(* Logix 5000 project; controller HP_SSC01hv vendor 1 type 14 code 158 rev 32.11; software revision 32.03; part 4 of 15 *)
(* tags used below, declared in another part *)
   A_C1_0422 : ALIAS FOR C1_Warning.22;
   A_C1_0423 : ALIAS FOR C1_Warning.23;
   A_C1_0425 : ALIAS FOR C1_Warning.25;
   A_C1_0426 : ALIAS FOR C1_Warning.26;
   C1_32HourTimers : TIMER[8];
   C1_ActualPositionMOD60 : REAL;
   C1_All_DLY_OK : BOOL;
   C1_Brake_Daily_ok : BOOL;
   C1_BrakeReleaseSelected : BOOL;
   C1_BrakeTestExpireTime : DINT;
   C1_BrakeTestExpireTimeTemp : DINT;
   C1_BrakeTestFailed : BOOL;
   C1_BrakeTestMessageNumber : DINT;
   C1_BrakeTestSelected : BOOL;
   C1_BrakeTestSequence : DINT;
   C1_BrakeTestWarning : BOOL;
   C1_DistanceToEvac : REAL;
   C1_Dump_OK : BOOL;
   C1_DumpValveReleaseSelected : BOOL;
   C1_DumpValveTestExpireTime : DINT;
   C1_DumpValveTestExpireTimeTemp : DINT;
   C1_DumpValveTestSelected : BOOL;
   C1_DumpValveTestSequence : DINT;
   C1_EvacPosition : REAL;
   C1_EvacPositionMOD60 : REAL;
   C1_ExcecutePBHoldTimer : TIMER;
   C1_FaultStandard : DINT;
   C1_GoNearOnPathDelay : TIMER;
   C1_GoToEvacMAM01 : MOTION_INSTRUCTION;
   C1_GoToOnPathMAM01 : MOTION_INSTRUCTION;
   C1_GoToOnPathMAM02 : MOTION_INSTRUCTION;
   C1_Home_OK : BOOL;
   C1_Homed : BOOL;
   C1_HomeExpireTime : DINT;
   C1_HomeExpireTimeTemp : DINT;
   C1_HomeSequence : DINT;
   C1_JogForwardFastSelected : BOOL;
   C1_JogForwardSlowSelected : BOOL;
   C1_JogReverseFastSelected : BOOL;
   C1_JogReverseSlowSelected : BOOL;
   C1_LubricationMessageNumber : DINT;
   C1_LubricationOnTimer : TIMER;
   C1_LubricationOverrideSelected : BOOL;
   C1_MAFR : MOTION_INSTRUCTION;
   C1_MAG : MOTION_INSTRUCTION;
   C1_MAJDeceleration : REAL;
   C1_MAS : MOTION_INSTRUCTION;
   C1_MASR : MOTION_INSTRUCTION;
   C1_Oiler : ALIAS FOR C1_RIO_AENT:O.Data[2].1;
   C1_OIT_BrakeRelease : BOOL;
   C1_OIT_BrakeReleaseDisplay : BOOL;
   C1_OIT_BrakeTest : BOOL;
   C1_OIT_BrakeTestDisplay : BOOL;
   C1_OIT_Command : DINT;
   C1_OIT_Current : DINT;
   C1_OIT_DumpValveRelease : BOOL;
   C1_OIT_DumpValveReleaseDisplay : BOOL;
   C1_OIT_DumpValveTest : BOOL;
   C1_OIT_DumpValveTestDisplay : BOOL;
   C1_OIT_FaultsExist : BOOL;
   C1_OIT_HomeCountDown : DINT;
   C1_OIT_JogForwardFast : BOOL;
   C1_OIT_JogForwardFastDisplay : BOOL;
   C1_OIT_JogForwardSlow : BOOL;
   C1_OIT_JogForwardSlowDisplay : BOOL;
   C1_OIT_JogReverseFast : BOOL;
   C1_OIT_JogReverseFastDisplay : BOOL;
   C1_OIT_JogReverseSlow : BOOL;
   C1_OIT_JogReverseSlowDisplay : BOOL;
   C1_OIT_JogStopDisplay : BOOL;
   C1_OIT_LubricationOverride : BOOL;
   C1_OIT_LubricationOverrideDisplay : BOOL;
   C1_OIT_PathError : DINT;
   C1_OIT_PathIndicatorHigh : DINT;
   C1_OIT_PathIndicatorLow : DINT;
   C1_OIT_WarningsExist : BOOL;
   C1_OneTryToFixErrorONS : BOOL;
   C1_ONS : DINT;
   C1_RemoteBrakeAndHomeSequence : DINT;
   C1_RemoteBrakeAndHomeSequenceAlarms : DINT;
   C1_RemoteBrakeAndHomeSequenceAlarmTimer : TIMER[32];
   C1_RemoteBrakeAndHomeSequenceONS : BOOL;
   C1_RemoteBrakeTestCMD : BOOL;
   C1_RemoteDumpTestCMD : BOOL;
   C1_RemoteHomeCMD : BOOL;
   C1_RemoteScreenMessageNumber : DINT;
   C1_RemoteSequenceDelay : TIMER[8];
   C1_RevolutionCounter : COUNTER;
   C1_ServoActionStatusOnDelay : TIMER;
   C1_TargetPositionError : REAL;
   C1_TargetPositionErrorTest : REAL;
   C1_Warning : DINT;
   MasterClockCopyMAS_Stop1 : MOTION_INSTRUCTION;
   MasterClockCopyMAS_Stop2 : MOTION_INSTRUCTION;
   MasterClockLocal : AXIS_VIRTUAL;
   none : BOOL;
   RCS_CMD_Auto_TON : TIMER;
   RCS_MasterClockLocalTagetDegrees : REAL;
   S_C1_FaultReset : BOOL;
   S_C1_FaultSafety : DINT;
   S_C1_ModeLocal : BOOL;
   S_C1_ModeRemote : BOOL;
   S_C1_MSTOP_InputOK : BOOL;
   S_C1_NearOnPath : BOOL;
   S_C1_NearOnPathHi : DINT;
   S_C1_NearOnPathLow : DINT;
   S_C1_OffPath : BOOL;
   S_C1_OnPath : BOOL;
   S_C1_PathError : DINT;
   S_RCS_MotionCMD_BrakeTest : BOOL;
   S_RCS_MotionCMD_Evac : BOOL;
   S_RCS_MotionCMD_GoNearOnPath : BOOL;
(* Carousel1, continued *)

ROUTINE C145_Lubrication   (* ladder *)
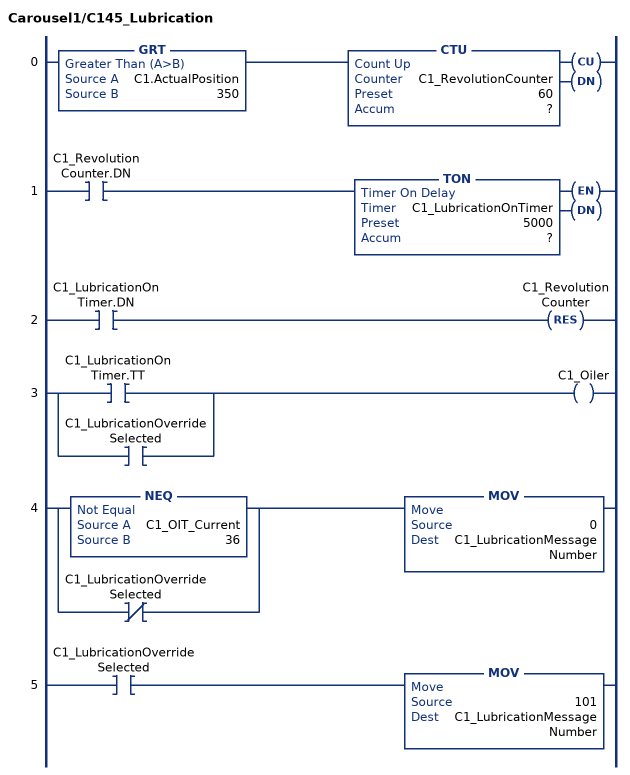
   0: GRT(C1.ActualPosition,350)CTU(C1_RevolutionCounter,?,?);
   1: XIC(C1_RevolutionCounter.DN)TON(C1_LubricationOnTimer,?,?);
   2: XIC(C1_LubricationOnTimer.DN)RES(C1_RevolutionCounter);
   3: [XIC(C1_LubricationOnTimer.TT) ,XIC(C1_LubricationOverrideSelected) ]OTE(C1_Oiler);
   4: [NEQ(C1_OIT_Current,36) ,XIO(C1_LubricationOverrideSelected) ]MOV(0,C1_LubricationMessageNumber);
   5: XIC(C1_LubricationOverrideSelected)MOV(101,C1_LubricationMessageNumber);
END_ROUTINE

ROUTINE C150_OIT   (* ladder *)
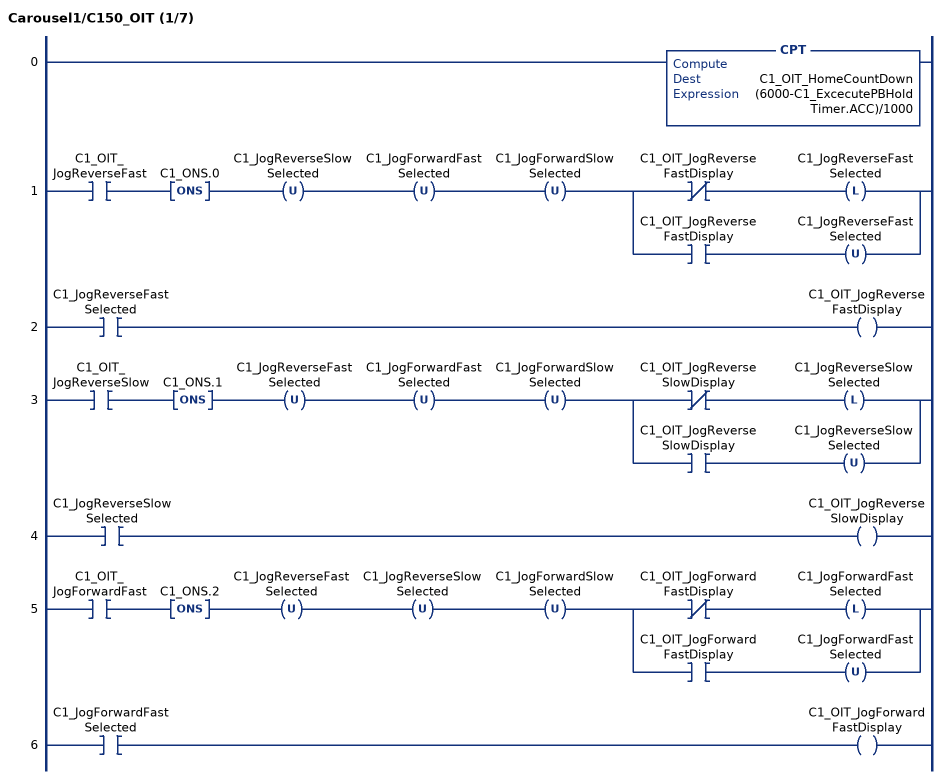
   0: CPT(C1_OIT_HomeCountDown,(6000-C1_ExcecutePBHoldTimer.ACC)/1000);
   1: XIC(C1_OIT_JogReverseFast)ONS(C1_ONS.0)OTU(C1_JogReverseSlowSelected)OTU(C1_JogForwardFastSelected)OTU(C1_JogForwardSlowSelected)[XIO(C1_OIT_JogReverseFastDisplay) OTL(C1_JogReverseFastSelected) ,XIC(C1_OIT_JogReverseFastDisplay) OTU(C1_JogReverseFastSelected) ];
   2: XIC(C1_JogReverseFastSelected)OTE(C1_OIT_JogReverseFastDisplay);
   3: XIC(C1_OIT_JogReverseSlow)ONS(C1_ONS.1)OTU(C1_JogReverseFastSelected)OTU(C1_JogForwardFastSelected)OTU(C1_JogForwardSlowSelected)[XIO(C1_OIT_JogReverseSlowDisplay) OTL(C1_JogReverseSlowSelected) ,XIC(C1_OIT_JogReverseSlowDisplay) OTU(C1_JogReverseSlowSelected) ];
   4: XIC(C1_JogReverseSlowSelected)OTE(C1_OIT_JogReverseSlowDisplay);
   5: XIC(C1_OIT_JogForwardFast)ONS(C1_ONS.2)OTU(C1_JogReverseFastSelected)OTU(C1_JogReverseSlowSelected)OTU(C1_JogForwardSlowSelected)[XIO(C1_OIT_JogForwardFastDisplay) OTL(C1_JogForwardFastSelected) ,XIC(C1_OIT_JogForwardFastDisplay) OTU(C1_JogForwardFastSelected) ];
   6: XIC(C1_JogForwardFastSelected)OTE(C1_OIT_JogForwardFastDisplay);
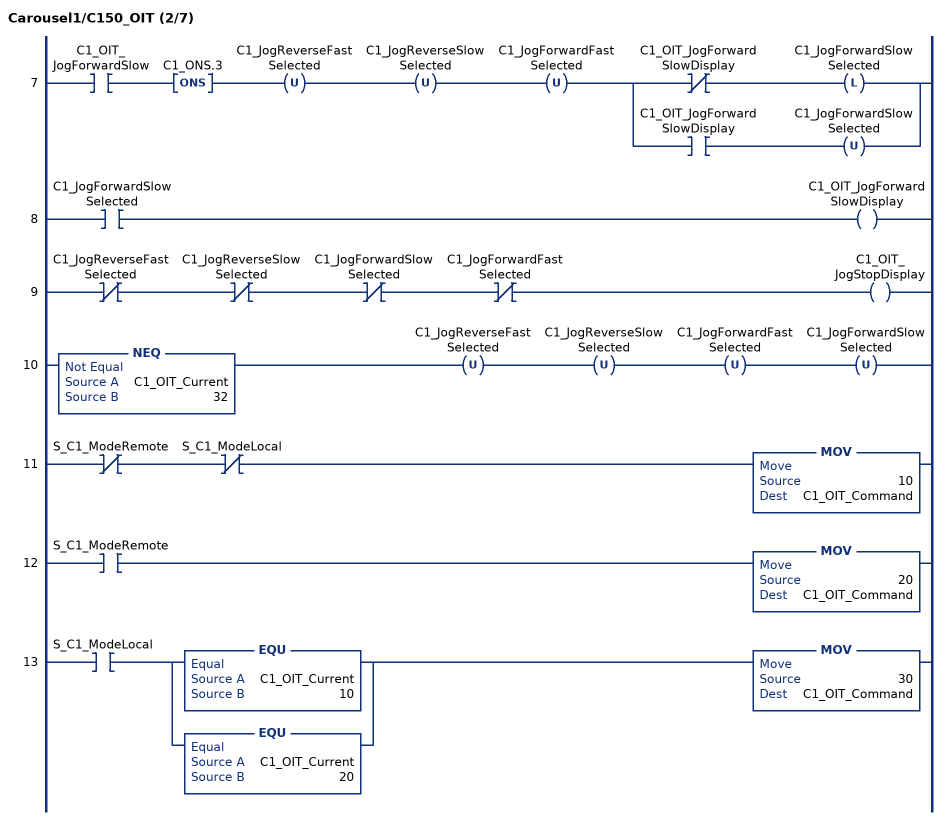
   7: XIC(C1_OIT_JogForwardSlow)ONS(C1_ONS.3)OTU(C1_JogReverseFastSelected)OTU(C1_JogReverseSlowSelected)OTU(C1_JogForwardFastSelected)[XIO(C1_OIT_JogForwardSlowDisplay) OTL(C1_JogForwardSlowSelected) ,XIC(C1_OIT_JogForwardSlowDisplay) OTU(C1_JogForwardSlowSelected) ];
   8: XIC(C1_JogForwardSlowSelected)OTE(C1_OIT_JogForwardSlowDisplay);
   9: XIO(C1_JogReverseFastSelected)XIO(C1_JogReverseSlowSelected)XIO(C1_JogForwardSlowSelected)XIO(C1_JogForwardFastSelected)OTE(C1_OIT_JogStopDisplay);
   10: NEQ(C1_OIT_Current,32)OTU(C1_JogReverseFastSelected)OTU(C1_JogReverseSlowSelected)OTU(C1_JogForwardFastSelected)OTU(C1_JogForwardSlowSelected);
   11: XIO(S_C1_ModeRemote)XIO(S_C1_ModeLocal)MOV(10,C1_OIT_Command);
   12: XIC(S_C1_ModeRemote)MOV(20,C1_OIT_Command);
   13: XIC(S_C1_ModeLocal)[EQU(C1_OIT_Current,10) ,EQU(C1_OIT_Current,20) ]MOV(30,C1_OIT_Command);
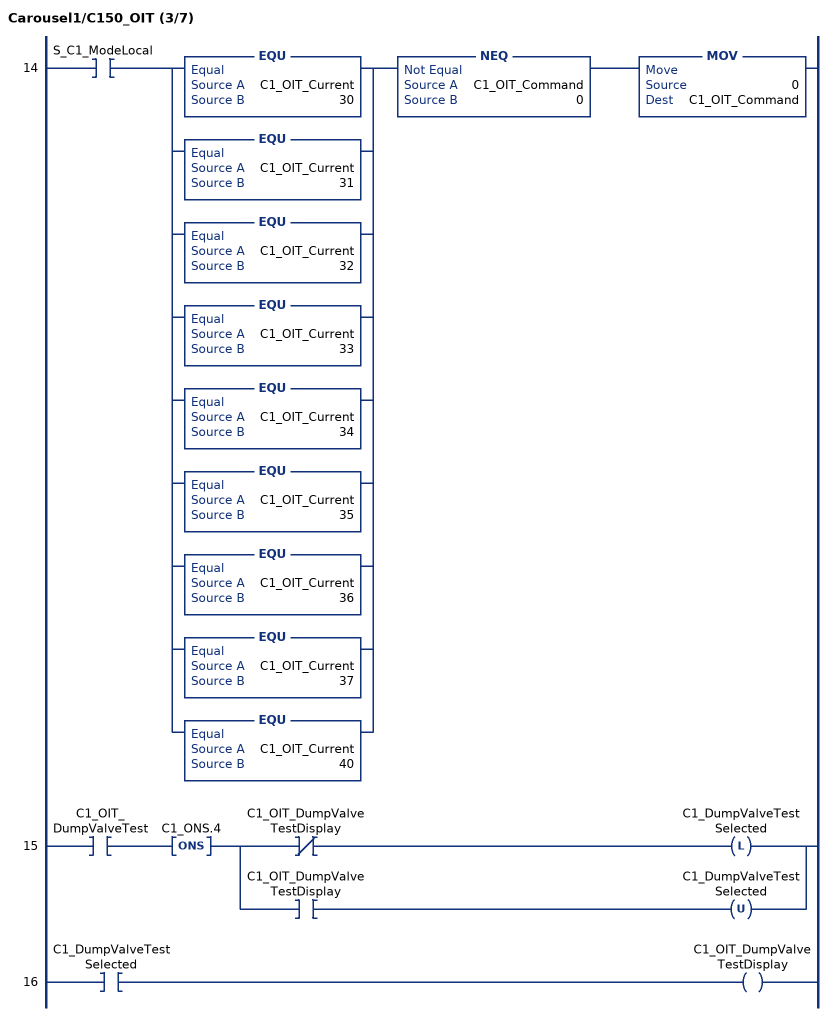
   14: XIC(S_C1_ModeLocal)[EQU(C1_OIT_Current,30) ,EQU(C1_OIT_Current,31) ,EQU(C1_OIT_Current,32) ,EQU(C1_OIT_Current,33) ,EQU(C1_OIT_Current,34) ,EQU(C1_OIT_Current,35) ,EQU(C1_OIT_Current,36) ,EQU(C1_OIT_Current,37) ,EQU(C1_OIT_Current,40) ]NEQ(C1_OIT_Command,0)MOV(0,C1_OIT_Command);
   15: XIC(C1_OIT_DumpValveTest)ONS(C1_ONS.4)[XIO(C1_OIT_DumpValveTestDisplay) OTL(C1_DumpValveTestSelected) ,XIC(C1_OIT_DumpValveTestDisplay) OTU(C1_DumpValveTestSelected) ];
   16: XIC(C1_DumpValveTestSelected)OTE(C1_OIT_DumpValveTestDisplay);
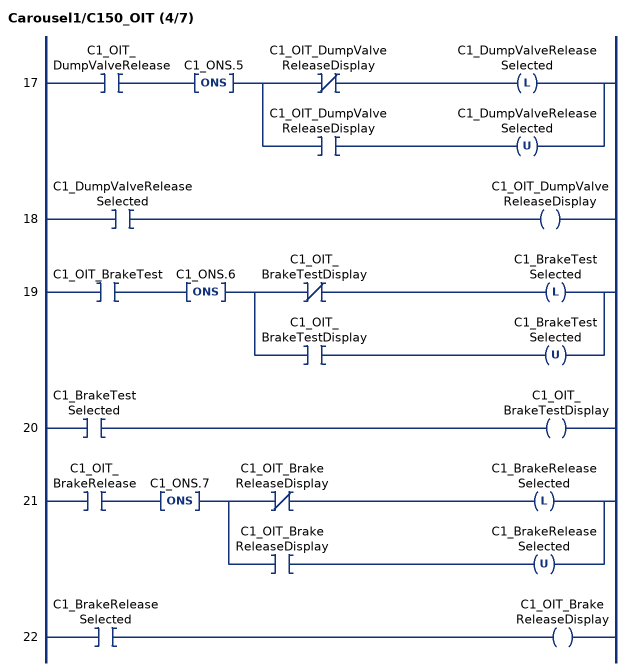
   17: XIC(C1_OIT_DumpValveRelease)ONS(C1_ONS.5)[XIO(C1_OIT_DumpValveReleaseDisplay) OTL(C1_DumpValveReleaseSelected) ,XIC(C1_OIT_DumpValveReleaseDisplay) OTU(C1_DumpValveReleaseSelected) ];
   18: XIC(C1_DumpValveReleaseSelected)OTE(C1_OIT_DumpValveReleaseDisplay);
   19: XIC(C1_OIT_BrakeTest)ONS(C1_ONS.6)[XIO(C1_OIT_BrakeTestDisplay) OTL(C1_BrakeTestSelected) ,XIC(C1_OIT_BrakeTestDisplay) OTU(C1_BrakeTestSelected) ];
   20: XIC(C1_BrakeTestSelected)OTE(C1_OIT_BrakeTestDisplay);
   21: XIC(C1_OIT_BrakeRelease)ONS(C1_ONS.7)[XIO(C1_OIT_BrakeReleaseDisplay) OTL(C1_BrakeReleaseSelected) ,XIC(C1_OIT_BrakeReleaseDisplay) OTU(C1_BrakeReleaseSelected) ];
   22: XIC(C1_BrakeReleaseSelected)OTE(C1_OIT_BrakeReleaseDisplay);
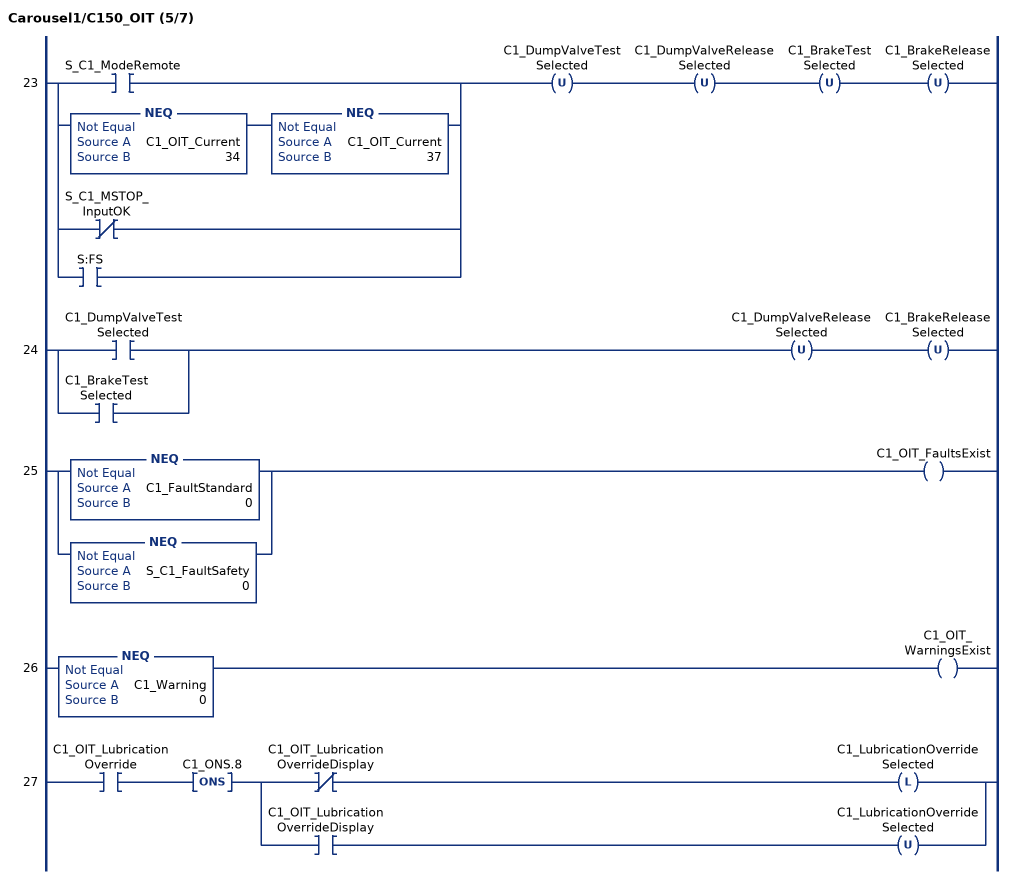
   23: [XIC(S_C1_ModeRemote) ,NEQ(C1_OIT_Current,34) NEQ(C1_OIT_Current,37) ,XIO(S_C1_MSTOP_InputOK) ,XIC(S:FS) ]OTU(C1_DumpValveTestSelected)OTU(C1_DumpValveReleaseSelected)OTU(C1_BrakeTestSelected)OTU(C1_BrakeReleaseSelected);
   24: [XIC(C1_DumpValveTestSelected) ,XIC(C1_BrakeTestSelected) ]OTU(C1_DumpValveReleaseSelected)OTU(C1_BrakeReleaseSelected);
   25: [NEQ(C1_FaultStandard,0) ,NEQ(S_C1_FaultSafety,0) ]OTE(C1_OIT_FaultsExist);
   26: NEQ(C1_Warning,0)OTE(C1_OIT_WarningsExist);
   27: XIC(C1_OIT_LubricationOverride)ONS(C1_ONS.8)[XIO(C1_OIT_LubricationOverrideDisplay) OTL(C1_LubricationOverrideSelected) ,XIC(C1_OIT_LubricationOverrideDisplay) OTU(C1_LubricationOverrideSelected) ];
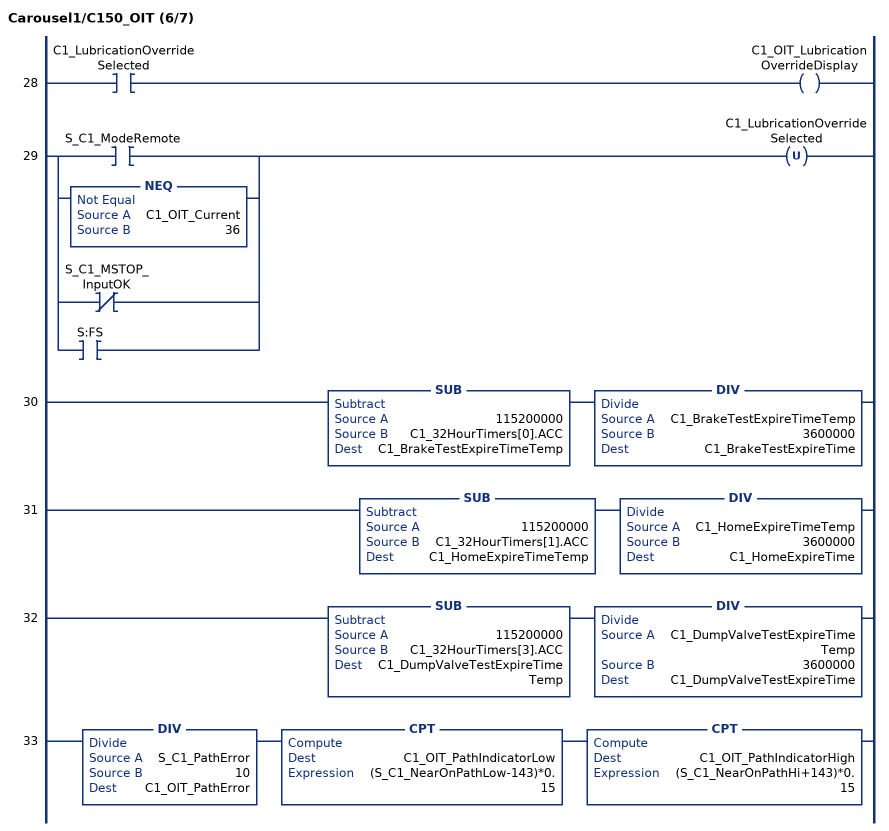
   28: XIC(C1_LubricationOverrideSelected)OTE(C1_OIT_LubricationOverrideDisplay);
   29: [XIC(S_C1_ModeRemote) ,NEQ(C1_OIT_Current,36) ,XIO(S_C1_MSTOP_InputOK) ,XIC(S:FS) ]OTU(C1_LubricationOverrideSelected);
   30: SUB(115200000,C1_32HourTimers[0].ACC,C1_BrakeTestExpireTimeTemp)DIV(C1_BrakeTestExpireTimeTemp,3600000,C1_BrakeTestExpireTime);
   31: SUB(115200000,C1_32HourTimers[1].ACC,C1_HomeExpireTimeTemp)DIV(C1_HomeExpireTimeTemp,3600000,C1_HomeExpireTime);
   32: SUB(115200000,C1_32HourTimers[3].ACC,C1_DumpValveTestExpireTimeTemp)DIV(C1_DumpValveTestExpireTimeTemp,3600000,C1_DumpValveTestExpireTime);
   33: DIV(S_C1_PathError,10,C1_OIT_PathError)CPT(C1_OIT_PathIndicatorLow,(S_C1_NearOnPathLow-143)*0.15)CPT(C1_OIT_PathIndicatorHigh,(S_C1_NearOnPathHi+143)*0.15);
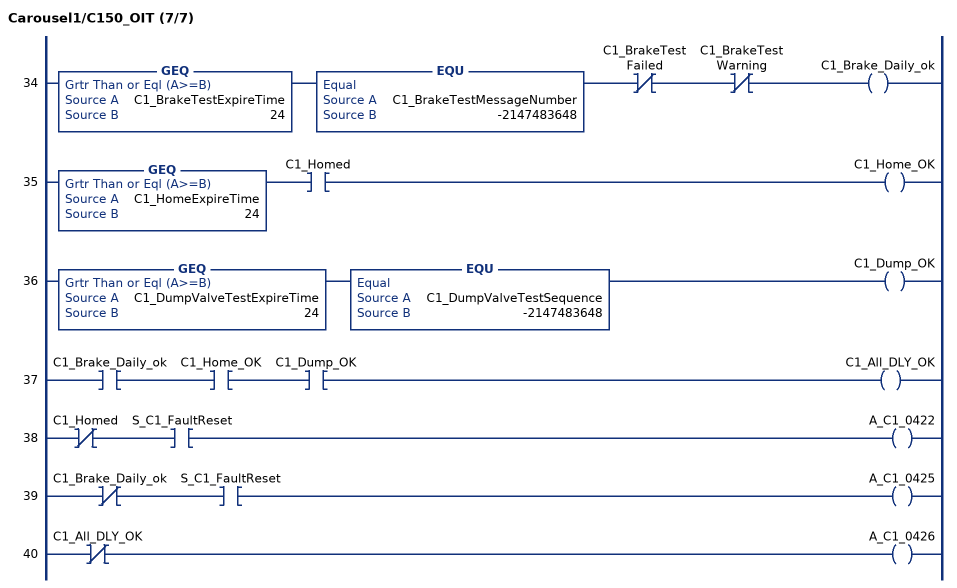
   34: GEQ(C1_BrakeTestExpireTime,24)EQU(C1_BrakeTestMessageNumber,-2147483648)XIO(C1_BrakeTestFailed)XIO(C1_BrakeTestWarning)OTE(C1_Brake_Daily_ok);
   35: GEQ(C1_HomeExpireTime,24)XIC(C1_Homed)OTE(C1_Home_OK);
   36: GEQ(C1_DumpValveTestExpireTime,24)EQU(C1_DumpValveTestSequence,-2147483648)OTE(C1_Dump_OK);
   37: XIC(C1_Brake_Daily_ok)XIC(C1_Home_OK)XIC(C1_Dump_OK)OTE(C1_All_DLY_OK);
   38: XIO(C1_Homed)XIC(S_C1_FaultReset)OTE(A_C1_0422);
   39: XIO(C1_Brake_Daily_ok)XIC(S_C1_FaultReset)OTE(A_C1_0425);
   40: XIO(C1_All_DLY_OK)OTE(A_C1_0426);
END_ROUTINE

ROUTINE C155_Remote   (* ladder *)
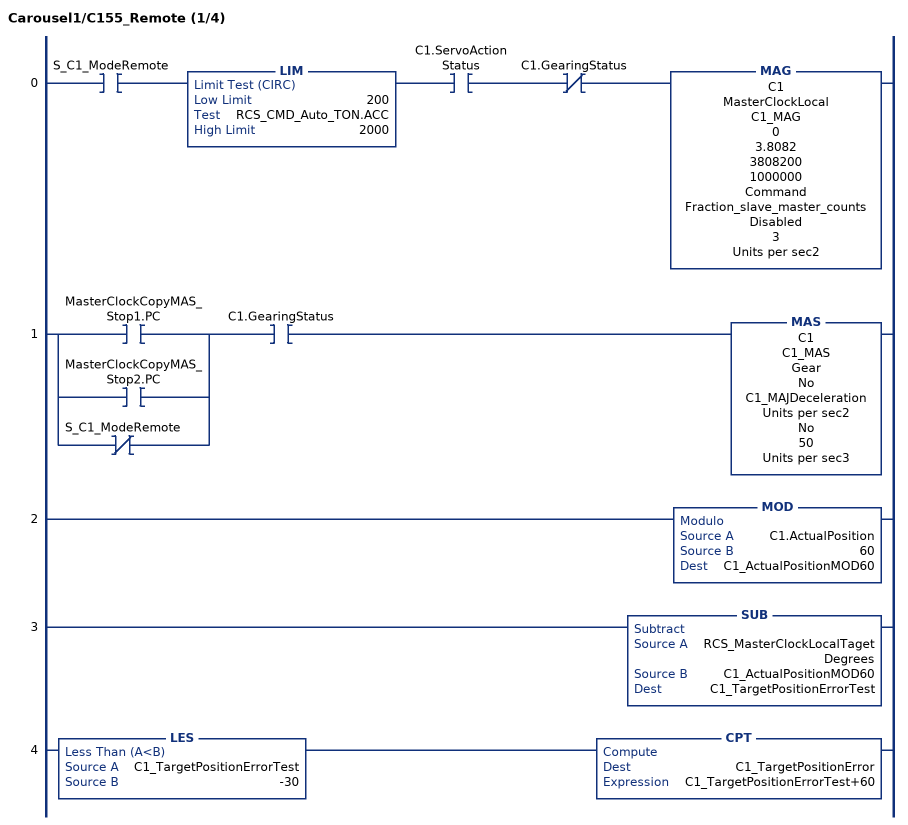
   0: XIC(S_C1_ModeRemote)LIM(200,RCS_CMD_Auto_TON.ACC,2000)XIC(C1.ServoActionStatus)XIO(C1.GearingStatus)MAG(C1,MasterClockLocal,C1_MAG,0,3.8082,3808200,1000000,Command,Fraction_slave_master_counts,Disabled,3,Units per sec2);
   1: [XIC(MasterClockCopyMAS_Stop1.PC) ,XIC(MasterClockCopyMAS_Stop2.PC) ,XIO(S_C1_ModeRemote) ]XIC(C1.GearingStatus)MAS(C1,C1_MAS,Gear,No,C1_MAJDeceleration,Units per sec2,No,50,Units per sec3);
   2: MOD(C1.ActualPosition,60,C1_ActualPositionMOD60);
   3: SUB(RCS_MasterClockLocalTagetDegrees,C1_ActualPositionMOD60,C1_TargetPositionErrorTest);
   4: LES(C1_TargetPositionErrorTest,-30)CPT(C1_TargetPositionError,C1_TargetPositionErrorTest+60);
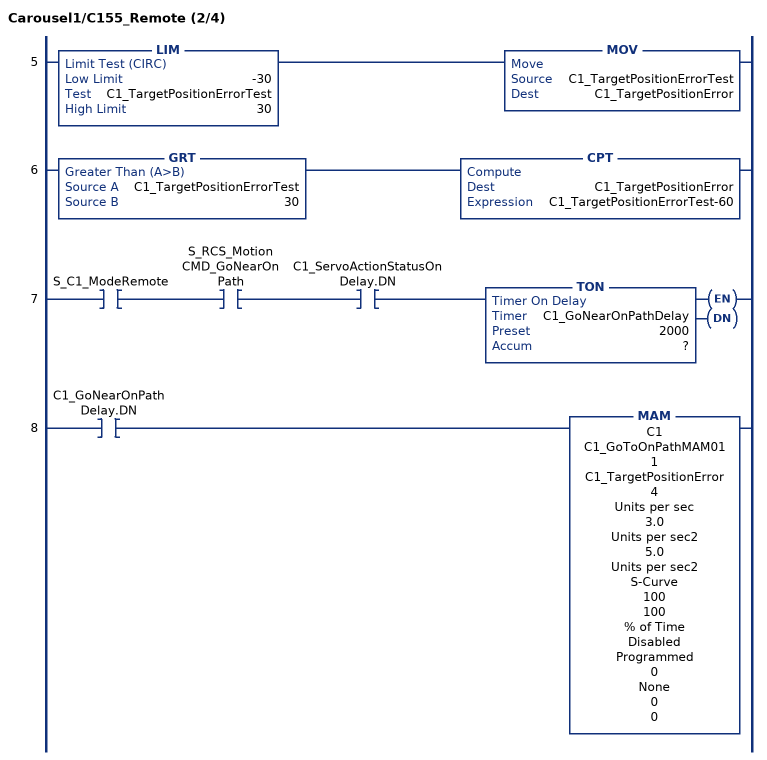
   5: LIM(-30,C1_TargetPositionErrorTest,30)MOV(C1_TargetPositionErrorTest,C1_TargetPositionError);
   6: GRT(C1_TargetPositionErrorTest,30)CPT(C1_TargetPositionError,C1_TargetPositionErrorTest-60);
   7: XIC(S_C1_ModeRemote)XIC(S_RCS_MotionCMD_GoNearOnPath)XIC(C1_ServoActionStatusOnDelay.DN)TON(C1_GoNearOnPathDelay,?,?);
   8: XIC(C1_GoNearOnPathDelay.DN)MAM(C1,C1_GoToOnPathMAM01,1,C1_TargetPositionError,4,Units per sec,3.0,Units per sec2,5.0,Units per sec2,S-Curve,100,100,% of Time,Disabled,Programmed,0,None,0,0);
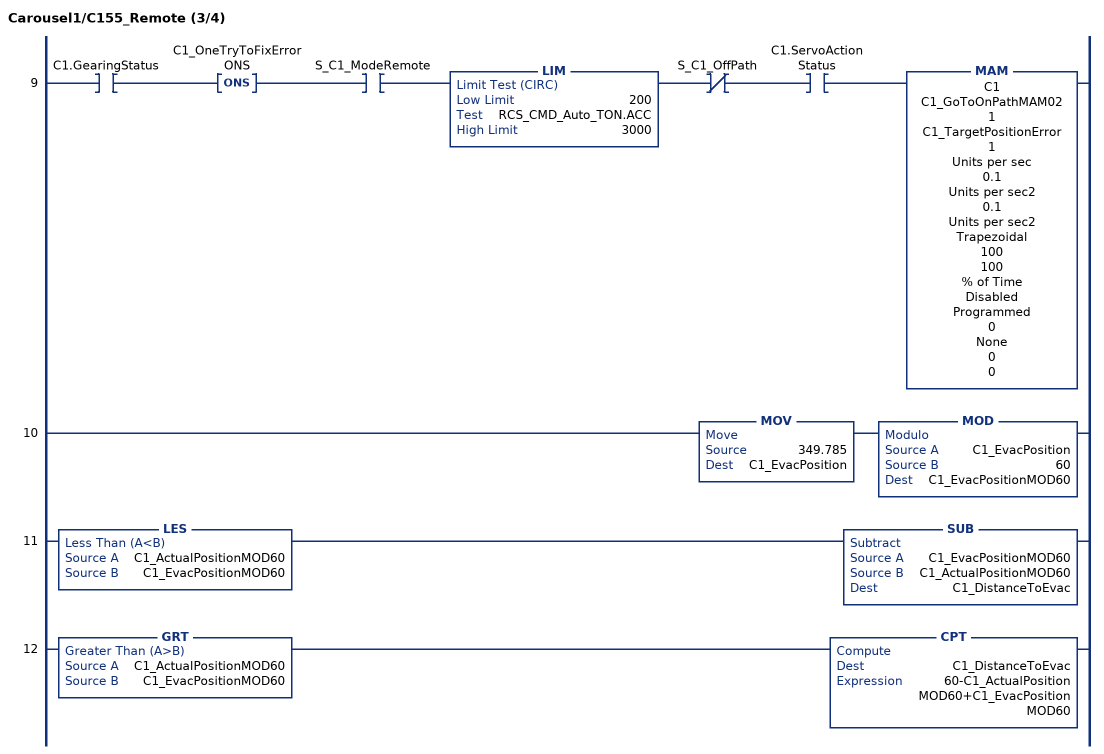
   9: XIC(C1.GearingStatus)ONS(C1_OneTryToFixErrorONS)XIC(S_C1_ModeRemote)LIM(200,RCS_CMD_Auto_TON.ACC,3000)XIO(S_C1_OffPath)XIC(C1.ServoActionStatus)MAM(C1,C1_GoToOnPathMAM02,1,C1_TargetPositionError,1,Units per sec,0.1,Units per sec2,0.1,Units per sec2,Trapezoidal,100,100,% of Time,Disabled,Programmed,0,None,0,0);
   10: MOV(349.785,C1_EvacPosition)MOD(C1_EvacPosition,60,C1_EvacPositionMOD60);
   11: LES(C1_ActualPositionMOD60,C1_EvacPositionMOD60)SUB(C1_EvacPositionMOD60,C1_ActualPositionMOD60,C1_DistanceToEvac);
   12: GRT(C1_ActualPositionMOD60,C1_EvacPositionMOD60)CPT(C1_DistanceToEvac,60-C1_ActualPositionMOD60+C1_EvacPositionMOD60);
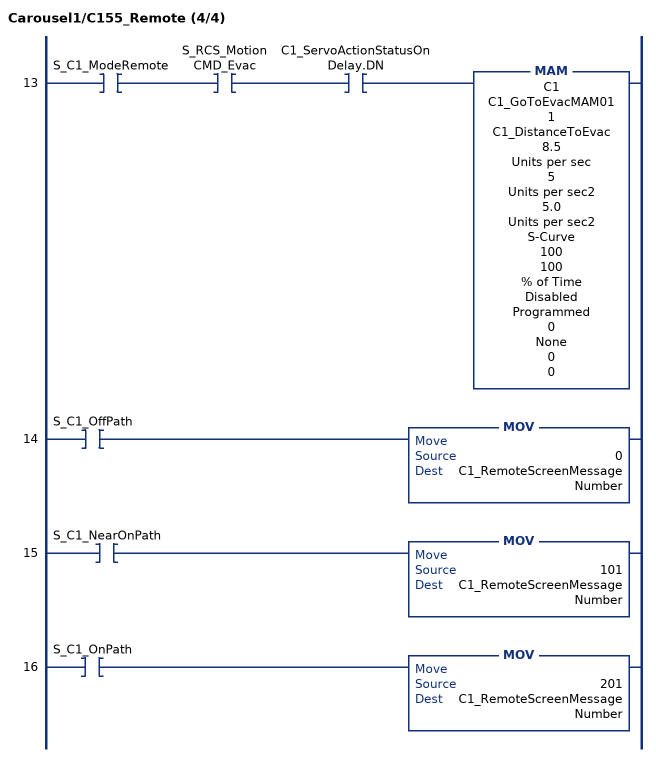
   13: XIC(S_C1_ModeRemote)XIC(S_RCS_MotionCMD_Evac)XIC(C1_ServoActionStatusOnDelay.DN)MAM(C1,C1_GoToEvacMAM01,1,C1_DistanceToEvac,8.5,Units per sec,5,Units per sec2,5.0,Units per sec2,S-Curve,100,100,% of Time,Disabled,Programmed,0,None,0,0);
   14: XIC(S_C1_OffPath)MOV(0,C1_RemoteScreenMessageNumber);
   15: XIC(S_C1_NearOnPath)MOV(101,C1_RemoteScreenMessageNumber);
   16: XIC(S_C1_OnPath)MOV(201,C1_RemoteScreenMessageNumber);
END_ROUTINE

ROUTINE C160_RemoteBrakeAndHome   (* ladder *)
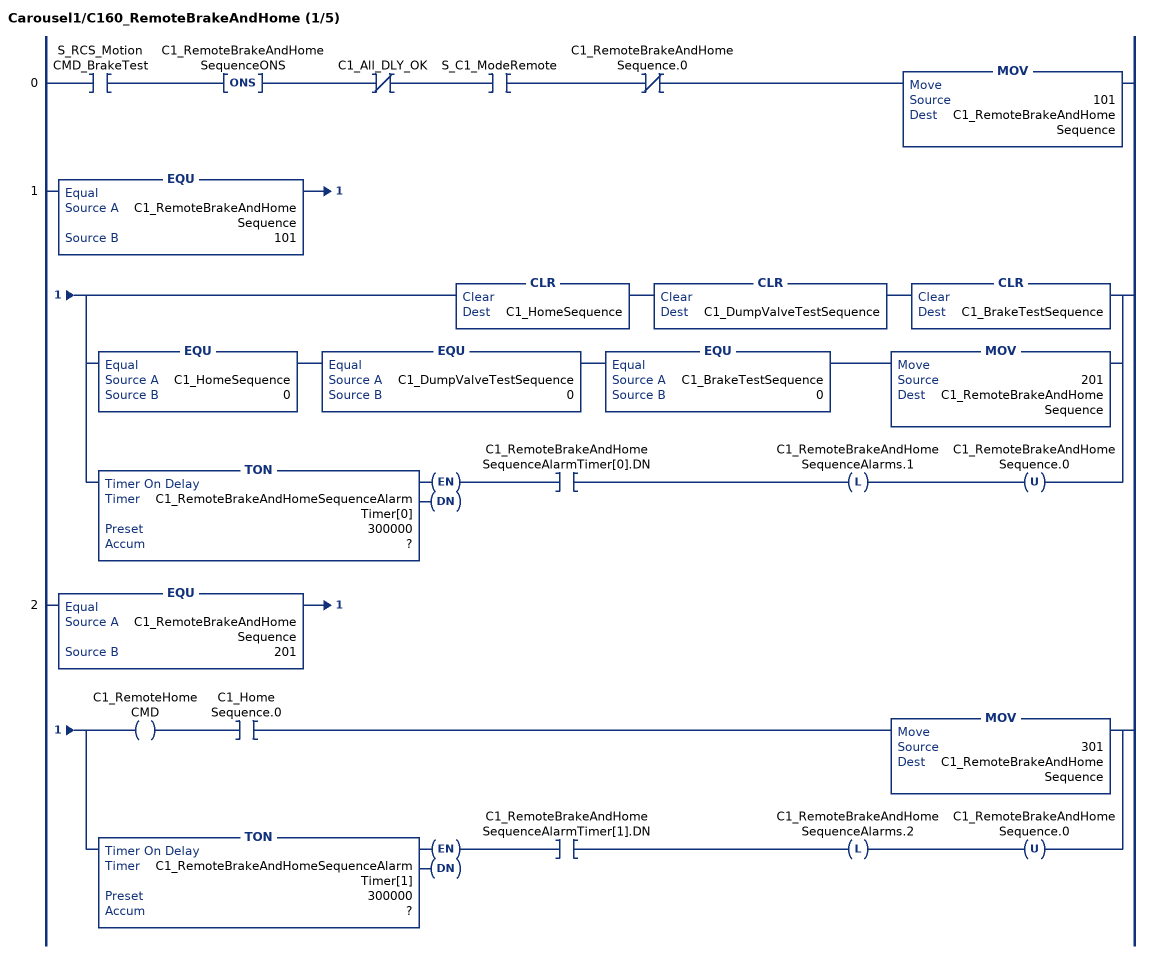
   0: XIC(S_RCS_MotionCMD_BrakeTest)ONS(C1_RemoteBrakeAndHomeSequenceONS)XIO(C1_All_DLY_OK)XIC(S_C1_ModeRemote)XIO(C1_RemoteBrakeAndHomeSequence.0)MOV(101,C1_RemoteBrakeAndHomeSequence);
   1: EQU(C1_RemoteBrakeAndHomeSequence,101)[CLR(C1_HomeSequence) CLR(C1_DumpValveTestSequence) CLR(C1_BrakeTestSequence) ,EQU(C1_HomeSequence,0) EQU(C1_DumpValveTestSequence,0) EQU(C1_BrakeTestSequence,0) MOV(201,C1_RemoteBrakeAndHomeSequence) ,TON(C1_RemoteBrakeAndHomeSequenceAlarmTimer[0],?,?) XIC(C1_RemoteBrakeAndHomeSequenceAlarmTimer[0].DN) OTL(C1_RemoteBrakeAndHomeSequenceAlarms.1) OTU(C1_RemoteBrakeAndHomeSequence.0) ];
   2: EQU(C1_RemoteBrakeAndHomeSequence,201)[OTE(C1_RemoteHomeCMD) XIC(C1_HomeSequence.0) MOV(301,C1_RemoteBrakeAndHomeSequence) ,TON(C1_RemoteBrakeAndHomeSequenceAlarmTimer[1],?,?) XIC(C1_RemoteBrakeAndHomeSequenceAlarmTimer[1].DN) OTL(C1_RemoteBrakeAndHomeSequenceAlarms.2) OTU(C1_RemoteBrakeAndHomeSequence.0) ];
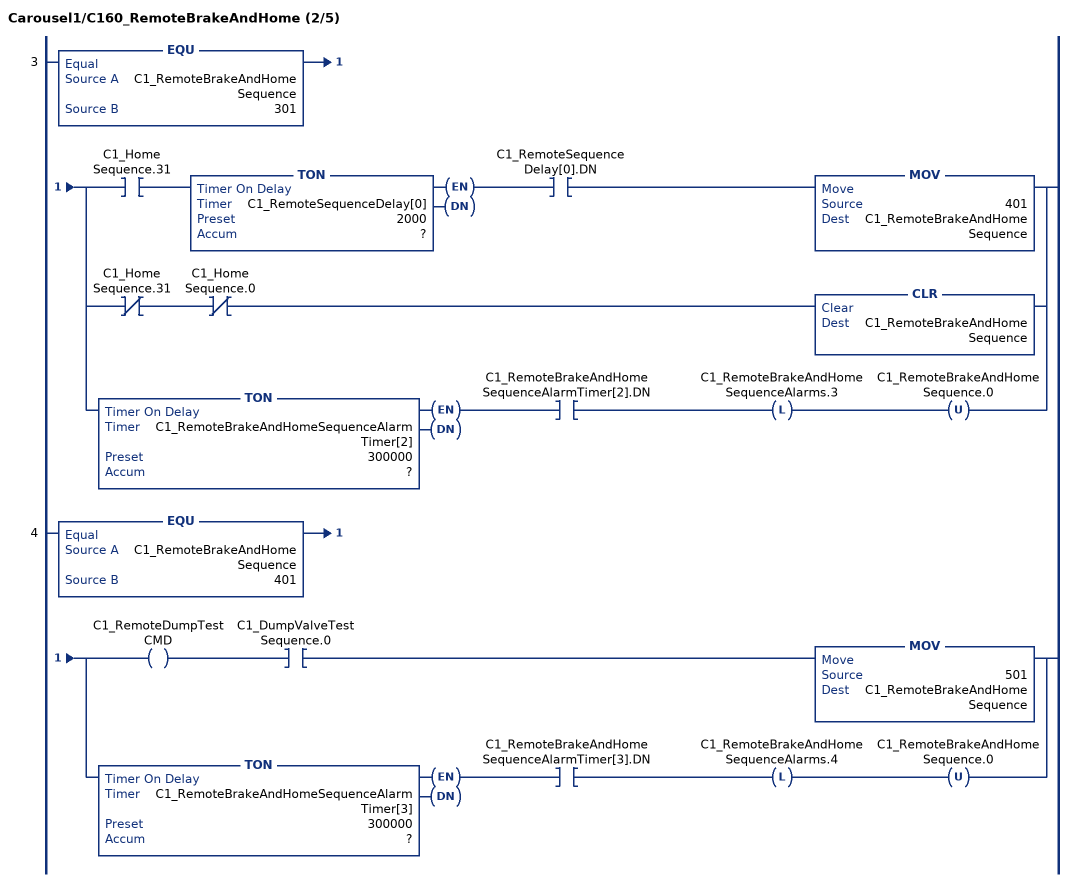
   3: EQU(C1_RemoteBrakeAndHomeSequence,301)[XIC(C1_HomeSequence.31) TON(C1_RemoteSequenceDelay[0],?,?) XIC(C1_RemoteSequenceDelay[0].DN) MOV(401,C1_RemoteBrakeAndHomeSequence) ,XIO(C1_HomeSequence.31) XIO(C1_HomeSequence.0) CLR(C1_RemoteBrakeAndHomeSequence) ,TON(C1_RemoteBrakeAndHomeSequenceAlarmTimer[2],?,?) XIC(C1_RemoteBrakeAndHomeSequenceAlarmTimer[2].DN) OTL(C1_RemoteBrakeAndHomeSequenceAlarms.3) OTU(C1_RemoteBrakeAndHomeSequence.0) ];
   4: EQU(C1_RemoteBrakeAndHomeSequence,401)[OTE(C1_RemoteDumpTestCMD) XIC(C1_DumpValveTestSequence.0) MOV(501,C1_RemoteBrakeAndHomeSequence) ,TON(C1_RemoteBrakeAndHomeSequenceAlarmTimer[3],?,?) XIC(C1_RemoteBrakeAndHomeSequenceAlarmTimer[3].DN) OTL(C1_RemoteBrakeAndHomeSequenceAlarms.4) OTU(C1_RemoteBrakeAndHomeSequence.0) ];
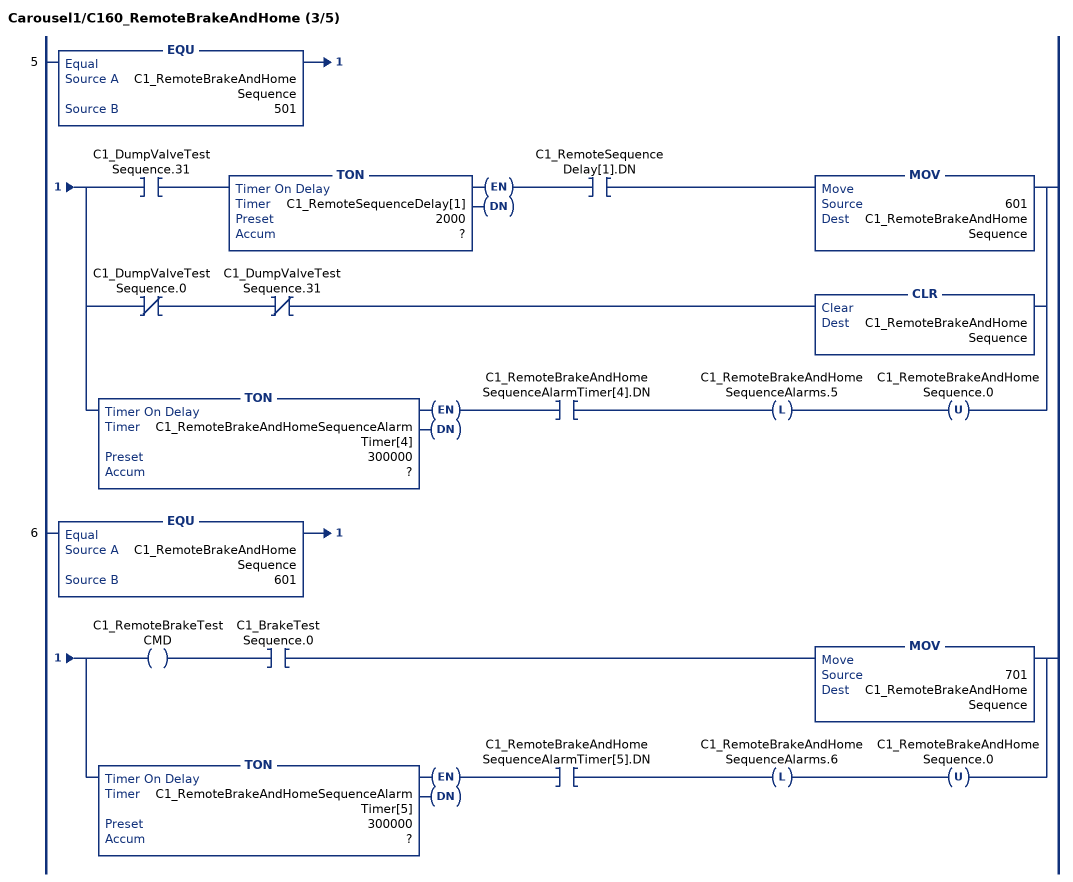
   5: EQU(C1_RemoteBrakeAndHomeSequence,501)[XIC(C1_DumpValveTestSequence.31) TON(C1_RemoteSequenceDelay[1],?,?) XIC(C1_RemoteSequenceDelay[1].DN) MOV(601,C1_RemoteBrakeAndHomeSequence) ,XIO(C1_DumpValveTestSequence.0) XIO(C1_DumpValveTestSequence.31) CLR(C1_RemoteBrakeAndHomeSequence) ,TON(C1_RemoteBrakeAndHomeSequenceAlarmTimer[4],?,?) XIC(C1_RemoteBrakeAndHomeSequenceAlarmTimer[4].DN) OTL(C1_RemoteBrakeAndHomeSequenceAlarms.5) OTU(C1_RemoteBrakeAndHomeSequence.0) ];
   6: EQU(C1_RemoteBrakeAndHomeSequence,601)[OTE(C1_RemoteBrakeTestCMD) XIC(C1_BrakeTestSequence.0) MOV(701,C1_RemoteBrakeAndHomeSequence) ,TON(C1_RemoteBrakeAndHomeSequenceAlarmTimer[5],?,?) XIC(C1_RemoteBrakeAndHomeSequenceAlarmTimer[5].DN) OTL(C1_RemoteBrakeAndHomeSequenceAlarms.6) OTU(C1_RemoteBrakeAndHomeSequence.0) ];
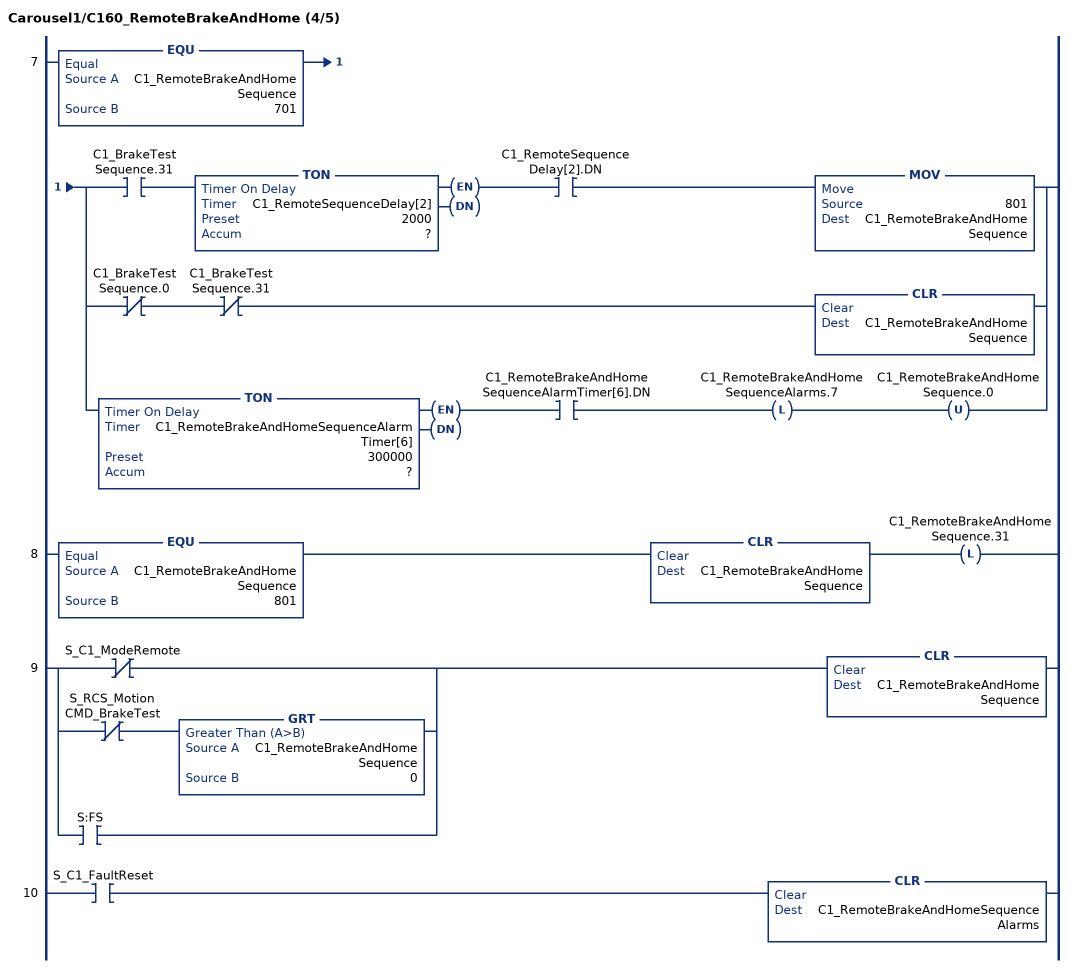
   7: EQU(C1_RemoteBrakeAndHomeSequence,701)[XIC(C1_BrakeTestSequence.31) TON(C1_RemoteSequenceDelay[2],?,?) XIC(C1_RemoteSequenceDelay[2].DN) MOV(801,C1_RemoteBrakeAndHomeSequence) ,XIO(C1_BrakeTestSequence.0) XIO(C1_BrakeTestSequence.31) CLR(C1_RemoteBrakeAndHomeSequence) ,TON(C1_RemoteBrakeAndHomeSequenceAlarmTimer[6],?,?) XIC(C1_RemoteBrakeAndHomeSequenceAlarmTimer[6].DN) OTL(C1_RemoteBrakeAndHomeSequenceAlarms.7) OTU(C1_RemoteBrakeAndHomeSequence.0) ];
   8: EQU(C1_RemoteBrakeAndHomeSequence,801)CLR(C1_RemoteBrakeAndHomeSequence)OTL(C1_RemoteBrakeAndHomeSequence.31);
   9: [XIO(S_C1_ModeRemote) ,XIO(S_RCS_MotionCMD_BrakeTest) GRT(C1_RemoteBrakeAndHomeSequence,0) ,XIC(S:FS) ]CLR(C1_RemoteBrakeAndHomeSequence);
   10: XIC(S_C1_FaultReset)CLR(C1_RemoteBrakeAndHomeSequenceAlarms);
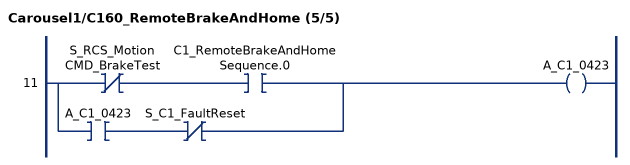
   11: [XIO(S_RCS_MotionCMD_BrakeTest) XIC(C1_RemoteBrakeAndHomeSequence.0) ,XIC(A_C1_0423) XIO(S_C1_FaultReset) ]OTE(A_C1_0423);
END_ROUTINE

ROUTINE C165_Reset   (* ladder *)
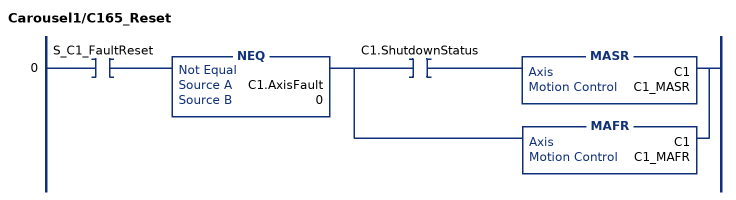
   0: XIC(S_C1_FaultReset)NEQ(C1.AxisFault,0)[XIC(C1.ShutdownStatus) MASR(C1,C1_MASR) ,MAFR(C1,C1_MAFR) ];
END_ROUTINE
END_PROGRAM
